SYSTEM DispenserMachineIncomplete (* Dispenser *)
  (* Standard: 61499-1 *)
  (* Version 0.4, 2009-03-05, JHC, Holobloc Inc., Deleted Application. *)
  (* Version 0.3, 2003-12-05, JHC, Rockwell Automation, Renamed from NEWSYSTEM. *)
  (* Version 0.2, 2002-11-05, JHC, Rockwell Automation, Fixed missing (empty) FBD in Application. *)
  (* Version 0.1, 2002-01-17, JHC, Rockwell Automation, Minor cleanup *)
  (* Version 0.0, 2000-05-27, JHC, Rockwell Automation *)
  DEVICE CoinsDetectorDevice : FRAME_DEVICE(BOUNDS := [0,0,200,300])
    RESOURCE RES : VIEW_PANEL(SIZE := [10,15], DIA := 20)
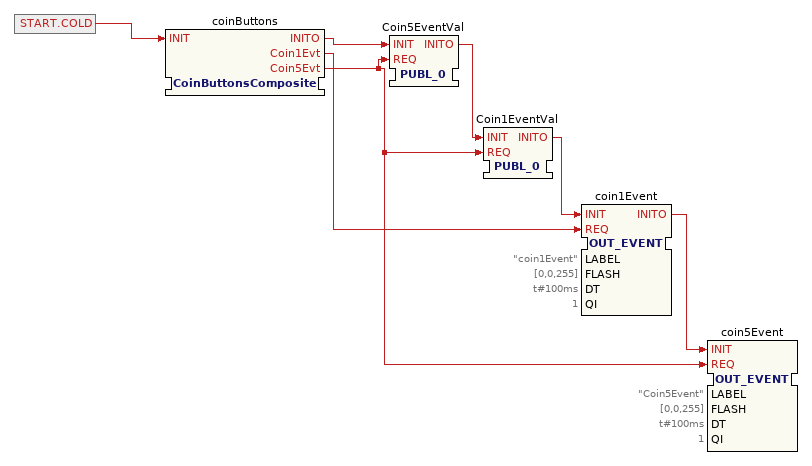
      FBS
        coin1Event : OUT_EVENT(LABEL := "coin1Event", FLASH := [0,0,255], DT := t#100ms, QI := 1);
        coin5Event : OUT_EVENT(LABEL := "Coin5Event", FLASH := [0,0,255], DT := t#100ms, QI := 1);
        Coin1EventVal : PUBL_0;
        Coin5EventVal : PUBL_0;
        coinButtons : CoinButtonsComposite;
      END_FBS
      EVENT_CONNECTIONS
        coin1Event.INITO TO coin5Event.INIT;
        Coin5EventVal.INITO TO Coin1EventVal.INIT;
        Coin1EventVal.INITO TO coin1Event.INIT;
        START.COLD TO coinButtons.INIT;
        coinButtons.INITO TO Coin5EventVal.INIT;
        coinButtons.Coin1Evt TO coin1Event.REQ;
        coinButtons.Coin5Evt TO coin5Event.REQ;
        coinButtons.Coin5Evt TO Coin5EventVal.REQ;
        coinButtons.Coin5Evt TO Coin1EventVal.REQ;
      END_CONNECTIONS
    END_RESOURCE
  END_DEVICE
  DEVICE HMIDevice : FRAME_DEVICE(BOUNDS := [0,0,200,300])
    RESOURCE RES : VIEW_PANEL(SIZE := [10,15], DIA := 20)
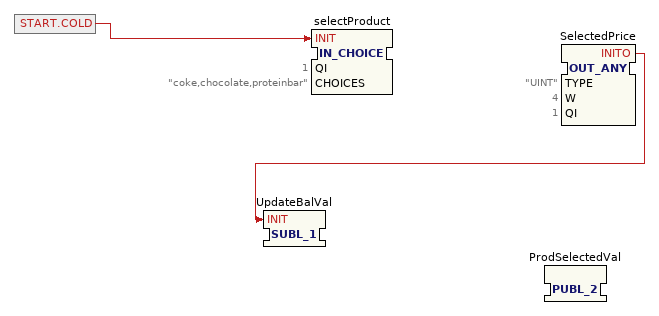
      FBS
        selectProduct : IN_CHOICE(QI := 1, CHOICES := "coke,chocolate,proteinbar");
        SelectedPrice : OUT_ANY(TYPE := "UINT", W := 4, QI := 1);
        UpdateBalVal : SUBL_1;
        ProdSelectedVal : PUBL_2;
      END_FBS
      EVENT_CONNECTIONS
        START.COLD TO selectProduct.INIT;
        SelectedPrice.INITO TO UpdateBalVal.INIT;
      END_CONNECTIONS
    END_RESOURCE
  END_DEVICE
  DEVICE ControlDevice : FRAME_DEVICE(BOUNDS := [0,0,200,300])
    RESOURCE RES : VIEW_PANEL(SIZE := [10,15], DIA := 20)
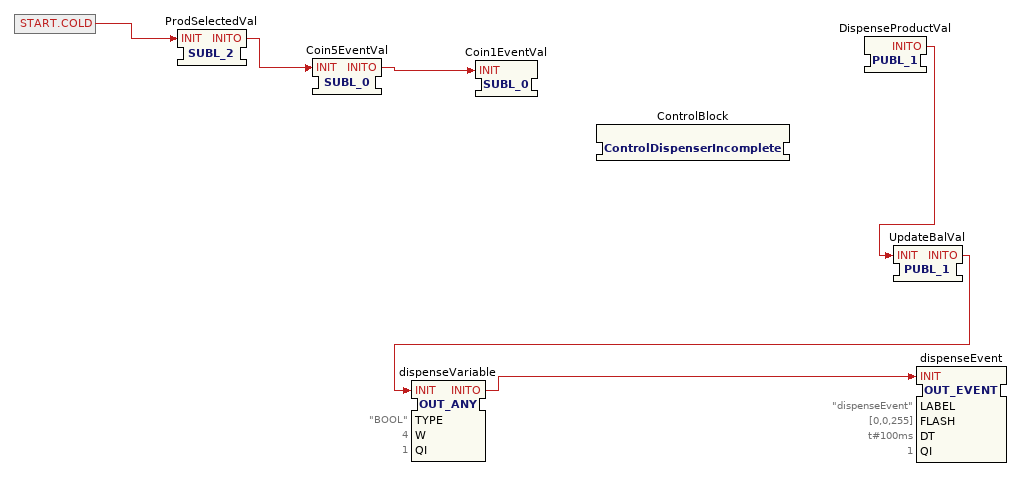
      FBS
        UpdateBalVal : PUBL_1;
        Coin5EventVal : SUBL_0;
        Coin1EventVal : SUBL_0;
        dispenseEvent : OUT_EVENT(LABEL := "dispenseEvent", FLASH := [0,0,255], DT := t#100ms, QI := 1);
        dispenseVariable : OUT_ANY(TYPE := "BOOL", W := 4, QI := 1);
        DispenseProductVal : PUBL_1;
        ProdSelectedVal : SUBL_2;
        ControlBlock : ControlDispenserIncomplete;
      END_FBS
      EVENT_CONNECTIONS
        Coin5EventVal.INITO TO Coin1EventVal.INIT;
        UpdateBalVal.INITO TO dispenseVariable.INIT;
        dispenseVariable.INITO TO dispenseEvent.INIT;
        START.COLD TO ProdSelectedVal.INIT;
        ProdSelectedVal.INITO TO Coin5EventVal.INIT;
        DispenseProductVal.INITO TO UpdateBalVal.INIT;
      END_CONNECTIONS
    END_RESOURCE
  END_DEVICE
  DEVICE DispenserMechanism : FRAME_DEVICE(BOUNDS := [0,0,200,300])
    RESOURCE RES : VIEW_PANEL(SIZE := [10,15], DIA := 20)
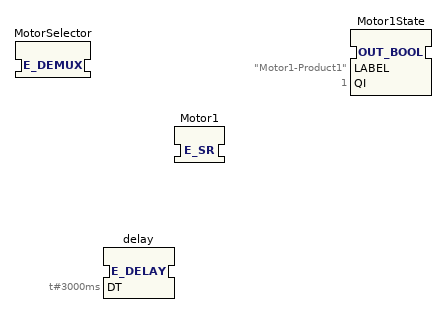
      FBS
        MotorSelector : E_DEMUX;
        delay : E_DELAY(DT := t#3000ms);
        Motor1 : E_SR;
        Motor1State : OUT_BOOL(LABEL := "Motor1-Product1", QI := 1);
      END_FBS
    END_RESOURCE
  END_DEVICE
END_SYSTEM
